FUNCTION_BLOCK EcMasterGetDeviceId IMPLEMENTS IEcTask
VAR_INPUT
END_VAR
VAR_OUTPUT
END_VAR
VAR
	iState : INT;
	getDeviceIdentity : Tc2_EtherCAT.FB_EcGetSlaveIdentity;
	_execute: BOOL;
	_done: BOOL;
	_busy: BOOL;
	_error: BOOL;
	_netId: AMSNETID;
END_VAR

CASE iState OF
	0:
		IF _execute THEN
			_done := FALSE;
			_busy := TRUE;
			_error := FALSE;
			getDeviceIdentity.bExecute := TRUE;
			IF getDeviceIdentity.bBusy THEN
				iState := 10;
				_execute := false;
			END_IF
		END_IF
	10:
		IF NOT getDeviceIdentity.bBusy THEN
			IF NOT getDeviceIdentity.bError THEN
				_done := TRUE;
			ELSE
				_error := TRUE;
			END_IF
			_busy := FALSE;
			getDeviceIdentity.bExecute := FALSE;
			iState := 0;
		END_IF
END_CASE

getDeviceIdentity(sNetId := Tc2_System.F_CreateAmsNetId(nIds := NetId));

{warning 'add method implementation '}
METHOD Abort : BOOL
getDeviceIdentity.bExecute := FALSE;
_busy := FALSE;
_execute := FALSE;
Abort := TRUE;
iState := 0;
END_METHOD

{warning 'add property implementation'}
PROPERTY Busy : BOOL
GET
Busy := _busy;
END_GET
END_PROPERTY

PROPERTY DeviceAddr : uint
GET
DeviceAddr := getDeviceIdentity.nSlaveAddr;
END_GET
SET
getDeviceIdentity.nSlaveAddr := DeviceAddr;
END_SET
END_PROPERTY

PROPERTY DeviceIdentity : ST_EcSlaveIdentity
GET
DeviceIdentity := getDeviceIdentity.identity;
END_GET
END_PROPERTY

{warning 'add property implementation'}
PROPERTY Done : BOOL
GET
Done := _done;
END_GET
END_PROPERTY

{warning 'add property implementation'}
PROPERTY Error : BOOL
GET
Error := _error;
END_GET
END_PROPERTY

{warning 'add method implementation '}
METHOD Execute : BOOL
IF NOT getDeviceIdentity.bBusy THEN
	Execute := _execute := true;
END_IF
END_METHOD

{warning 'add property implementation'}
PROPERTY NetID : amsnetid
GET
NetID := _netId;
END_GET
SET
_netId := NetID;
END_SET
END_PROPERTY

END_FUNCTION_BLOCK

(* stored: Version 1.1.0.1, ProductVersion 3.1.4024.11
   POU EcMasterGetDeviceId: Id {dc65c762-4ea8-4ac1-a513-61e5daa816cc}, SpecialFunc None
   Method Abort: Id {21b4edfa-8e91-4315-b900-f533312b3eb0}
   Property Busy: Id {3b2b0c65-f6a3-4fde-ac76-c5b9134394cb}
   Get Get: Id {33c462b1-e879-454c-a700-d1de5ed80c72}
   Property DeviceAddr: Id {f5624484-91d8-496f-90f4-c44328886d34}
   Get Get: Id {df1f344d-8d0d-4ada-a373-55768cd3e53e}
   Set Set: Id {19410178-6145-4d2d-bd8d-e9c7f0e330c9}
   Property DeviceIdentity: Id {7ca5304a-a3f3-48b0-a667-1fb78e203775}
   Get Get: Id {4b04ae76-ac66-4502-a228-c8e5aeb992db}
   Property Done: Id {b8c152fd-6732-4d88-9012-859b090a9a56}
   Get Get: Id {5fe7ad21-a30f-454a-af70-fbd1158b7cd8}
   Property Error: Id {16287692-7c3e-4de8-b023-2606442667fc}
   Get Get: Id {7acf5a3c-f31a-4a10-b6f1-70da9662731e}
   Method Execute: Id {9d3e3844-b26d-4288-a722-0f3f44081ca0}
   Property NetID: Id {0f681d85-42c4-432c-9217-1c654b4499b2}
   Get Get: Id {5cbf8ad9-a715-4d40-9d18-136724c5e48d}
   Set Set: Id {ecc78eda-61fe-415d-ab73-3022ef6da546} *)
